{attribute 'qualified_only'}
{attribute 'strict'}
TYPE E_AmpelPhase :
(
	INIT := 0,
	ROT,
	GRUEN,
	GELB,
	ROTGELB
);
END_TYPE

(* stored: Version 1.1.0.1, ProductVersion 3.1.4024.12
   DUT E_AmpelPhase: Id {4a04ad9d-b5ba-462a-8b8d-57ae1cd32cd1} *)
